FUNCTION_BLOCK fb_Counter
VAR_INPUT
	bActive		:	BOOL;
	bReset		:	BOOL;
END_VAR
VAR_OUTPUT
	iCounter	:	INT;
END_VAR
VAR
END_VAR

IF bActive THEN
	iCounter := iCounter + 1;
ELSE
	IF bReset THEN
		iCounter := 0;
	END_IF
END_IF

END_FUNCTION_BLOCK

(* stored: Version 1.1.0.1, ProductVersion 3.1.4024.12
   POU fb_Counter: Id {3946809f-9678-4f04-a4f2-dba97a9f3222}, SpecialFunc None *)
